// atan2(y,x)
FUNCTION F_atan2 : LREAL
VAR_INPUT
	y:	LREAL;
	x:	LREAL;
END_VAR
VAR
	atan2val:	LREAL;
END_VAR

IF (x > 0) THEN
	atan2val := ATAN(y/x);
ELSIF ((x < 0) AND (y >= 0)) THEN
	atan2val := ATAN(y/x) + GCL.C_PI;
ELSIF ((x < 0) AND (y < 0)) THEN
	atan2val := ATAN(y/x) - GCL.C_PI;
ELSIF ((x = 0) AND (y > 0)) THEN
	atan2val := GCL.C_PI2;
ELSIF ((x = 0) AND (y < 0)) THEN
	atan2val := -GCL.C_PI2;
ELSIF ((x = 0) AND (y = 0)) THEN
	atan2val := 1000;  //represents undefined
END_IF             

F_atan2	:= atan2val;

END_FUNCTION

(* stored: Version 1.1.0.1, ProductVersion 3.1.4022.9
   POU F_atan2: Id {a975d600-9d78-4379-9d76-f7bbd5a83222}, SpecialFunc None *)
